// ---- VISUs/PAGE_MAIN.TcVIS
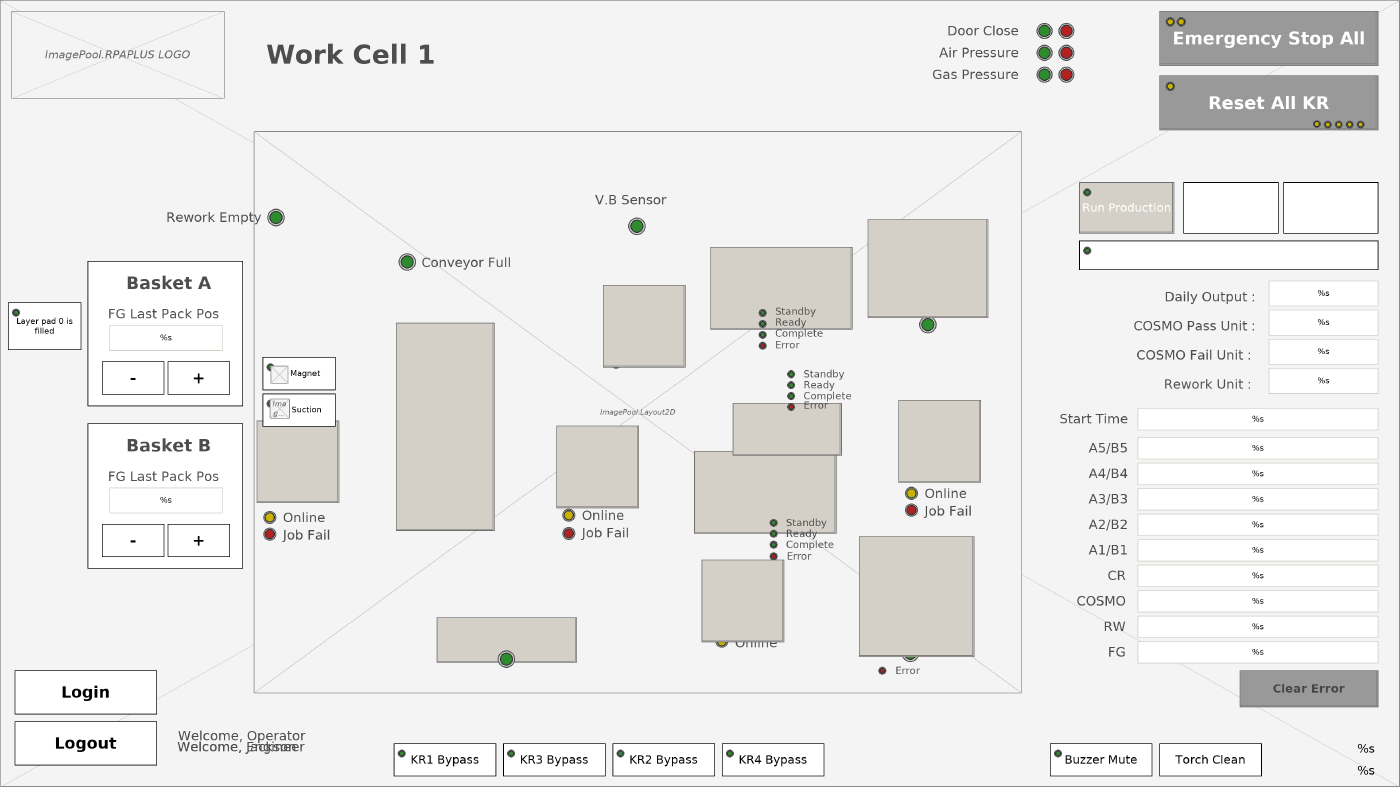
VISUALIZATION PAGE_MAIN  // 1920x1080
    Image (0,0 1920x1080), image: ImagePool.The-New-Silver-Backgrounds
    Frame (0,930 1920x150)
        shows Footer_Main()
        shows Footer_1()
    Frame (0,0 1920x225)
        shows Header()
    Label (362,45 650x60), "Work Cell 1"
    RoundedRectangle (1760,250 130x70), "Reset Production"
        OnMouseClick: OpenDialog Dialog=MSG_BOX_RESET, OpenModal=True, OpenCentered=True
    RoundedRectangle (20,990 195x60), "Logout"
        OnMouseClick: VisuUserMgmt Type=Logout
        OnMouseClick: execute {
            LOGFILE( sLogEvent	 := MSG.EVENT_BTN,
            		 sLogComp	 := MSG.COMP_HMI,
            		 sLogAction	 := MSG.ACTION_LOGOUT,
            	 	 logFlag	 := TRUE);
        }
    RoundedRectangle (20,920 195x60), "Login"
        tap MAIN.BTN_LOG
        OnMouseClick: VisuUserMgmt Type=Login
        OnMouseClick: execute {
            LOGFILE( sLogEvent	 := MSG.EVENT_BTN,
            		 sLogComp	 := MSG.COMP_HMI,
            		 sLogAction	 := MSG.ACTION_LOGIN,
            	 	 logFlag	 := TRUE);
        }
    Label (240,1005 200x40), "Welcome, Engineer"
    Label (240,1005 200x40), "Welcome, Jackson"
    Label (241,990 200x40), "Welcome, Operator"
    RoundedRectangle (120,358 213x199)
    Label (170,366 119x45), "Basket A"
    RoundedRectangle (140,496 85x45), "-"
        tap JIG.BasketA_Minus
        OnMouseClick: execute {
            LOGFILE( sLogEvent	 := MSG.EVENT_BTN,
            		 sLogComp	 := MSG.COMP_FG,
            		 sLogAction	 := MSG.ACTION_BSKTA_MINUS,
            	 	 logFlag	 := TRUE);
        }
    RoundedRectangle (230,496 85x45), "+"
        tap JIG.BasketA_Plus
        OnMouseClick: execute {
            LOGFILE( sLogEvent	 := MSG.EVENT_BTN,
            		 sLogComp	 := MSG.COMP_FG,
            		 sLogAction	 := MSG.ACTION_BSKTA_PLUS,
            	 	 logFlag	 := TRUE);
        }
    Textfield (150,446 155x35), "%s", text variable: GVL.Basket_A_Counter
    Label (145,416 173x30), "FG Last Pack Pos"
    RoundedRectangle (120,581 213x199)
    Label (170,589 119x45), "Basket B"
    RoundedRectangle (140,719 85x45), "-"
        tap JIG.BasketB_Minus
        OnMouseClick: execute {
            LOGFILE( sLogEvent	 := MSG.EVENT_BTN,
            		 sLogComp	 := MSG.COMP_FG,
            		 sLogAction	 := MSG.ACTION_BSKTA_MINUS,
            	 	 logFlag	 := TRUE);
        }
    RoundedRectangle (230,719 85x45), "+"
        tap JIG.BasketB_Plus
        OnMouseClick: execute {
            LOGFILE( sLogEvent	 := MSG.EVENT_BTN,
            		 sLogComp	 := MSG.COMP_FG,
            		 sLogAction	 := MSG.ACTION_BSKTB_PLUS,
            	 	 logFlag	 := TRUE);
        }
    Textfield (150,669 155x35), "%s", text variable: GVL.Basket_B_Counter
    Label (145,639 173x30), "FG Last Pack Pos"
    Image (348,180 1053x771), image: ImagePool.Layout2D
    Lamp1 (865,430 27x27), variable: KR3.bInBit[1,6], style: Lamp-Lamp1-Green
    Lamp1 (1010,815 27x27), variable: KR4.bInBit[1,6], style: Lamp-Lamp1-Green
    Lamp1 (1275,600 27x27), variable: KR5.bInBit[1,6], style: Lamp-Lamp1-Green
    Lamp1 (800,625 27x27), variable: KR2.bInBit[1,6], style: Lamp-Lamp1-Green
    Lamp1 (360,700 20x20), variable: KR1.KROnline, style: Lamp-Lamp1-Yellow
    Button (543,443 135x285)
        OnMouseClick: change screen: PAGE_CoolRack
        OnMouseClick: execute {
            LOGFILE( sLogEvent	 := MSG.EVENT_PAGE,
            		 sLogComp	 := MSG.COMP_CR,
            		 sLogAction	 := MSG.ACTION_COOLRACK,
            	 	 logFlag	 := TRUE);
        }
    Button (599,847 192x62)
        OnMouseClick: change screen: PAGE_COSMO
        OnMouseClick: execute {
            LOGFILE( sLogEvent	 := MSG.EVENT_PAGE,
            		 sLogComp	 := MSG.COMP_CM,
            		 sLogAction	 := MSG.ACTION_COSMO,
            	 	 logFlag	 := TRUE);
        }
    Lamp1 (681,891 27x27), variable: GVL.COSMO_Ready, style: Lamp-Lamp1-Green
    Lamp1 (860,297 27x27), variable: GVL.VibBowl_Ready, style: Lamp-Lamp1-Green
    Label (813,252 255x45), "V.B Sensor"
    Lamp1 (1259,432 27x27), variable: INFEED_RACK.IFRack_Ready, style: Lamp-Lamp1-Green
    Lamp1 (1235,883 27x27), variable: GVL.JIGC_Standby, style: Lamp-Lamp1-Green
    Button (1178,736 158x165)
        OnMouseClick: change screen: PAGE_TTorch
        OnMouseClick: execute {
            LOGFILE( sLogEvent	 := MSG.EVENT_PAGE,
            		 sLogComp	 := MSG.COMP_TT,
            		 sLogAction	 := MSG.ACTION_TT,
            	 	 logFlag	 := TRUE);
        }
    Button (974,339 195x113)
        OnMouseClick: change screen: PAGE_JIG_A
        OnMouseClick: execute {
            LOGFILE( sLogEvent	 := MSG.EVENT_PAGE,
            		 sLogComp	 := MSG.COMP_JIGA,
            		 sLogAction	 := MSG.ACTION_JIGA,
            	 	 logFlag	 := TRUE);
        }
    Button (952,619 195x113)
        OnMouseClick: change screen: PAGE_JIG_C
        OnMouseClick: execute {
            LOGFILE( sLogEvent	 := MSG.EVENT_PAGE,
            		 sLogComp	 := MSG.COMP_JIGC,
            		 sLogAction	 := MSG.ACTION_JIGC,
            	 	 logFlag	 := TRUE);
        }
    Button (1005,553 149x72)
        OnMouseClick: change screen: PAGE_JIG_B
        OnMouseClick: execute {
            LOGFILE( sLogEvent	 := MSG.EVENT_PAGE,
            		 sLogComp	 := MSG.COMP_JIGB,
            		 sLogAction	 := MSG.ACTION_JIGB,
            	 	 logFlag	 := TRUE);
        }
    Lamp1 (365,285 27x27), variable: GVL.Rework_Empty, style: Lamp-Lamp1-Green
    Lamp1 (545,346 27x27), variable: GVL.Conveyor_Full, style: Lamp-Lamp1-Green
    Label (225,276 146x45), "Rework Empty"
    Label (575,338 130x45), "Conveyor Full"
    Lamp1 (360,723 20x20), variable: KR1.bInBit[4,0], style: Lamp-Lamp1-Red
    Lamp1 (1240,690 20x20), variable: KR5.bInBit[4,7], style: Lamp-Lamp1-Red
    Lamp1 (770,722 20x20), variable: KR2.bInBit[3,4], style: Lamp-Lamp1-Red
    Lamp1 (395,633 27x27), variable: KR1.bInBit[1,6], style: Lamp-Lamp1-Green
    Label (385,722 80x25), "Job Fail"
    Label (385,698 80x25), "Online"
    Lamp1 (770,697 20x20), variable: KR2.KROnline, style: Lamp-Lamp1-Yellow
    Label (795,719 80x25), "Job Fail"
    Label (795,695 80x25), "Online"
    Lamp1 (1240,667 20x20), variable: KR5.KROnline, style: Lamp-Lamp1-Yellow
    Label (1265,689 80x25), "Job Fail"
    Label (1265,665 80x25), "Online"
    Lamp1 (835,487 20x20), variable: KR3.KROnline, style: Lamp-Lamp1-Yellow
    Label (860,485 80x25), "Online"
    Lamp1 (980,870 20x20), variable: KR4.KROnline, style: Lamp-Lamp1-Yellow
    Label (1005,870 80x25), "Online"
    Button (827,391 113x113)
        OnMouseClick: change screen: PAGE_KR3
        OnMouseClick: execute {
            LOGFILE( sLogEvent	 := MSG.EVENT_PAGE,
            		 sLogComp	 := MSG.COMP_KR3,
            		 sLogAction	 := MSG.ACTION_KR3,
            	 	 logFlag	 := TRUE);
        }
    Button (763,584 113x113)
        OnMouseClick: change screen: PAGE_KR2
        OnMouseClick: execute {
            LOGFILE( sLogEvent	 := MSG.EVENT_PAGE,
            		 sLogComp	 := MSG.COMP_KR2,
            		 sLogAction	 := MSG.ACTION_KR2,
            	 	 logFlag	 := TRUE);
        }
    Button (962,768 113x113)
        OnMouseClick: change screen: PAGE_KR4
        OnMouseClick: execute {
            LOGFILE( sLogEvent	 := MSG.EVENT_PAGE,
            		 sLogComp	 := MSG.COMP_KR4,
            		 sLogAction	 := MSG.ACTION_KR4,
            	 	 logFlag	 := TRUE);
        }
    Button (1232,549 113x113)
        OnMouseClick: change screen: PAGE_KR5
        OnMouseClick: execute {
            LOGFILE( sLogEvent	 := MSG.EVENT_PAGE,
            		 sLogComp	 := MSG.COMP_KR5,
            		 sLogAction	 := MSG.ACTION_KR5,
            	 	 logFlag	 := TRUE);
        }
    Button (352,577 113x113)
        OnMouseClick: change screen: PAGE_KR1_Tab
        OnMouseClick: execute {
            LOGFILE( sLogEvent	 := MSG.EVENT_PAGE,
            		 sLogComp	 := MSG.COMP_KR1,
            		 sLogAction	 := MSG.ACTION_KR1,
            	 	 logFlag	 := TRUE);
        }
    Label (1500,425 225x45), "COSMO Pass Unit :"
    Textfield (1740,425 150x35), "%s", text variable: GVL.Pass_Counter
    Textfield (1740,465 150x35), "%s", text variable: GVL.Fail_Counter
    Label (1500,465 225x45), "COSMO Fail Unit :"
    Textfield (1560,880 330x30), "%s", text variable: AUTO_MODE.processnameFG
    Group (1430,705 460x30)
        Textfield (130,0 330x30), "%s", text variable: AUTO_MODE.processnameA2
        Label (0,0 120x30), "A2/B2"
    Group (1430,740 460x30)
        Textfield (130,0 330x30), "%s", text variable: AUTO_MODE.processnameA1
        Label (0,0 120x30), "A1/B1"
    Textfield (1560,600 330x30), "%s", text variable: AUTO_MODE.processnameA5
    Label (1430,600 120x30), "A5/B5"
    Group (1430,635 460x30)
        Textfield (130,0 330x30), "%s", text variable: AUTO_MODE.processnameA4
        Label (0,0 120x30), "A4/B4"
    Group (1430,670 460x30)
        Textfield (130,0 330x30), "%s", text variable: AUTO_MODE.processnameA3
        Label (0,0 120x30), "A3/B3"
    Label (1472,880 75x30), "FG"
    Group (1472,845 418x30)
        Textfield (88,0 330x30), "%s", text variable: AUTO_MODE.processnameRW
        Label (0,0 75x30), "RW"
    Group (1472,775 418x30)
        Textfield (88,0 330x30), "%s", text variable: AUTO_MODE.processnameCR
        Label (0,0 75x30), "CR"
    Group (1455,810 435x30)
        Textfield (105,0 330x30), "%s", text variable: AUTO_MODE.processnameCOSMO
        Label (0,0 92x30), "COSMO"
    Lamp1 (1260,358 20x20), variable: INFEED_RACK.IFRack_Ready, style: Lamp-Lamp1-Yellow
    Button (1190,301 165x135)
        OnMouseClick: change screen: PAGE_InfeedRack
        OnMouseClick: execute {
            LOGFILE( sLogEvent	 := MSG.EVENT_PAGE,
            		 sLogComp	 := MSG.COMP_IR,
            		 sLogAction	 := MSG.ACTION_INFEEDRACK,
            	 	 logFlag	 := TRUE);
        }
    Label (1500,385 225x45), "Daily Output :"
    Textfield (1740,385 150x35), "%s", text variable: GVL.daily_output
    Label (1500,505 225x45), "Rework Unit :"
    Textfield (1740,505 150x35), "%s", text variable: GVL.Rework_Counter
    RoundedRectangle (1480,330 410x40), "Welding Mode"
        toggle SAFETY_SENSOR.WELDING_MODE
        OnMouseClick: execute {  }
    RoundedRectangle (1623,250 130x70), "Halt Production", input disabled if: MAIN.btnTorchClean
        OnMouseClick: execute {
            KR1.bOutBit[1,0]:= FALSE;
            KR2.bOutBit[1,0]:= FALSE;
            KR3.bOutBit[1,0]:= FALSE;
            KR4.bOutBit[1,0]:= FALSE;
            KR5.bOutBit[1,0]:= FALSE;
            LOGFILE( sLogEvent	 := MSG.EVENT_BTN,
            		 sLogComp	 := MSG.COMP_HMI,
            		 sLogAction	 := MSG.ACTION_STOP,
            	 	 logFlag	 := TRUE);
            AUTO_MODE.Halt_Production := TRUE;
            AUTO_MODE.AutoMode := False;
        }
    Button (1480,250 130x70), "Run Production", pressed state: AUTO_MODE.AutoMode, input disabled if: MAIN.btnTorchClean
        toggle AUTO_MODE.AutoMode
        OnMouseClick: execute {
            LOGFILE( sLogEvent	 := MSG.EVENT_BTN,
            		 sLogComp	 := MSG.COMP_HMI,
            		 sLogAction	 := MSG.ACTION_START,
            	 	 logFlag	 := TRUE);
            IF AUTO_MODE.AutoMode THEN
            	AUTO_MODE.Start_time := MAIN.fb_TimeStamp.SystemTime;
            END_IF
        }
    Lamp1 (1485,255 12x18), variable: AUTO_MODE.AutoMode, style: Lamp-Lamp1-Green
    Textfield (1560,560 330x30), "%s", text variable: AUTO_MODE.Start_time
    Label (1430,560 120x30), "Start Time"
    Lamp1 (1485,335 12x18), variable: SAFETY_SENSOR.WELDING_MODE, style: Lamp-Lamp1-Green
    Group (1250,20 225x105)
        Group (0,0 225x45)
            Label (0,0 150x45), "Door Close"
            Lamp1 (170,10 25x25), variable: SAFETY_SENSOR.SENSOR_SAFETY_DOOR_CLOSE, style: Lamp-Lamp1-Green
            Lamp1 (200,10 25x25), variable: not SAFETY_SENSOR.SENSOR_SAFETY_DOOR_CLOSE, style: Lamp-Lamp1-Red
        Label (0,30 150x45), "Air Pressure"
        Lamp1 (170,40 25x25), variable: SAFETY_SENSOR.SENSOR_AIR_PRESSURE_OK, style: Lamp-Lamp1-Green
        Lamp1 (200,40 25x25), variable: not SAFETY_SENSOR.SENSOR_AIR_PRESSURE_OK or SAFETY_SENSOR.SENSOR_AIR_PRESSURE_HIGH, style: Lamp-Lamp1-Red
        Label (0,60 150x45), "Gas Pressure"
        Lamp1 (170,70 25x25), variable: SAFETY_SENSOR.SENSOR_GAS_PRESSURE_OK, style: Lamp-Lamp1-Green
        Lamp1 (200,70 25x25), variable: not SAFETY_SENSOR.SENSOR_GAS_PRESSURE_OK or SAFETY_SENSOR.SENSOR_GAS_PRESSURE_HIGH, style: Lamp-Lamp1-Red
    Group (1079,506 100x45)
        Lamp1 (0,0 12x15), variable: GVL.JIGB_Standby, style: Lamp-Lamp1-Green
        Lamp1 (0,15 12x15), variable: GVL.JIGB_Ready, style: Lamp-Lamp1-Green
        Label (20,0 80x15), "Standby"
        Label (20,15 80x15), "Ready"
        Label (20,30 80x15), "Complete"
        Lamp1 (0,30 12x15), variable: GVL.JIGB_Complete, style: Lamp-Lamp1-Green
    Lamp1 (1040,422 12x15), variable: GVL.JIGA_Standby, style: Lamp-Lamp1-Green
    Lamp1 (1040,437 12x15), variable: GVL.JIGA_Ready, style: Lamp-Lamp1-Green
    Label (1060,420 80x15), "Standby"
    Label (1060,435 80x15), "Ready"
    Label (1060,450 80x15), "Complete"
    Lamp1 (1040,452 12x15), variable: GVL.JIGA_Complete, style: Lamp-Lamp1-Green
    Lamp1 (1055,710 12x15), variable: GVL.JIGC_Standby, style: Lamp-Lamp1-Green
    Lamp1 (1055,725 12x15), variable: GVL.JIGC_Ready, style: Lamp-Lamp1-Green
    Label (1075,710 80x15), "Standby"
    Label (1075,725 80x15), "Ready"
    Label (1075,740 80x15), "Complete"
    Lamp1 (1055,740 12x15), variable: GVL.JIGC_Complete, style: Lamp-Lamp1-Green
    Button (1700,920 190x50), "Clear Error", pressed state: MAIN.btn_Reset or MAIN.Reset_State
        toggle GVL.ClearError
        OnMouseClick: execute {
            LOGFILE( sLogEvent	 := MSG.EVENT_BTN,
            		 sLogComp	 := MSG.COMP_HMI,
            		 sLogAction	 := MSG.ACTION_CLEAR_ERROR,
            	 	 logFlag	 := TRUE);
        }
    Label (1060,466 80x15), "Error"
    Lamp1 (1040,467 12x15), variable: AUTO_MODE.JIGA_ErrorState, style: Lamp-Lamp1-Red
    Lamp1 (1079,551 12x15), variable: AUTO_MODE.JIGB_ErrorState, style: Lamp-Lamp1-Red
    Label (1099,549 80x15), "Error"
    Lamp1 (1055,756 12x15), variable: AUTO_MODE.JIGC_ErrorState, style: Lamp-Lamp1-Red
    Label (1076,756 80x15), "Error"
    Lamp1 (1204,913 12x15), variable: AUTO_MODE.TT_ErrorState, style: Lamp-Lamp1-Red
    Label (1225,913 80x15), "Error"
    RoundedRectangle (1590,1020 140x45), "Torch Clean"
        toggle MAIN.btnTorchClean
        OnMouseClick: execute {  }
    Group (1440,1020 140x45)
        RoundedRectangle (0,0 140x45), "Buzzer Mute"
            toggle TL.Buzzer_mute
            OnMouseClick: execute {  }
        Lamp1 (5,5 12x18), variable: TL.Buzzer_mute, style: Lamp-Lamp1-Green
    Group (840,1020 290x45)
        Group (150,0 140x45)
            RoundedRectangle (0,0 140x45), "KR4 Bypass"
                OnMouseClick: OpenDialog Dialog=MSG_KR4_BP, OpenModal=True, OpenCentered=True
            Lamp1 (5,5 12x18), variable: GVL.KR4_bypass, style: Lamp-Lamp1-Green
        RoundedRectangle (0,0 140x45), "KR2 Bypass"
            OnMouseClick: OpenDialog Dialog=MSG_KR2_BP, OpenModal=True, OpenCentered=True
        Lamp1 (5,5 12x18), variable: GVL.KR2_bypass, style: Lamp-Lamp1-Green
    RoundedRectangle (690,1020 140x45), "KR3 Bypass"
        OnMouseClick: OpenDialog Dialog=MSG_KR3_BP, OpenModal=True, OpenCentered=True
    Lamp1 (695,1025 12x18), variable: GVL.KR3_bypass, style: Lamp-Lamp1-Green
    RoundedRectangle (540,1020 140x45), "KR1 Bypass"
        OnMouseClick: OpenDialog Dialog=MSG_KR1_BP, OpenModal=True, OpenCentered=True
    Lamp1 (545,1025 12x18), variable: GVL.KR1_bypass, style: Lamp-Lamp1-Green
    Group (360,490 100x45)
        RoundedRectangle (0,0 100x45), "Magnet"
            OnMouseClick: OpenDialog Dialog=MSG_EOAT, OpenModal=True, OpenCentered=True
        Lamp1 (5,5 12x18), variable: GVL.KR1_EOAT_FILL, style: Lamp-Lamp1-Green
        Image (11,12 24x24), image: ImagePool.001-resources
    Group (360,540 100x45)
        RoundedRectangle (0,0 100x45), "Suction"
            OnMouseClick: OpenDialog Dialog=MSG_EOAT_SUCTION, OpenModal=True, OpenCentered=True
        Lamp1 (5,5 12x18), variable: GVL.KR1_EOAT_SUCTION, style: Lamp-Lamp1-Green
        Image (10,7 27x27), angle 180, image: ImagePool.002-plunger
    RoundedRectangle (11,415 100x65), "Layer pad 0 is filled"
        toggle GVL.LAYERPAD0
    Lamp1 (16,420 12x18), variable: GVL.LAYERPAD0, style: Lamp-Lamp1-Green
END_VISUALIZATION

// ---- VISUs/PAGE_KR2.TcVIS
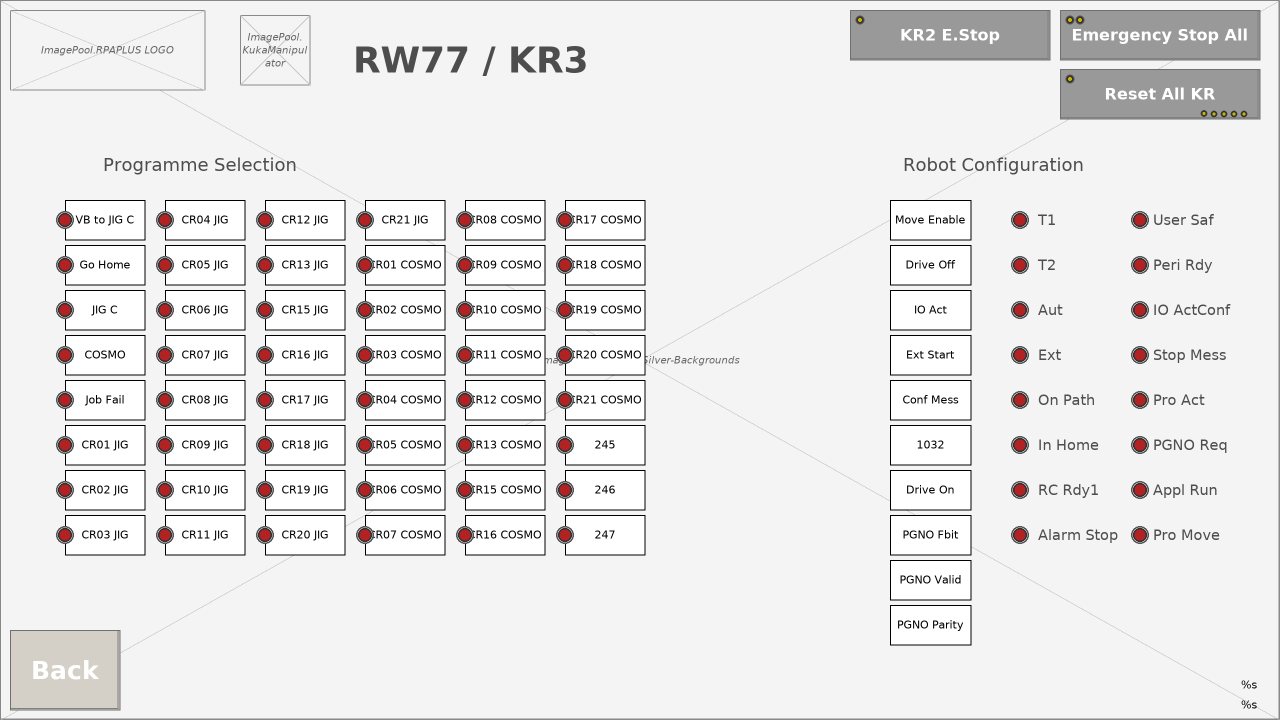
VISUALIZATION PAGE_KR2  // 1280x720
    Image (0,0 1280x720), image: ImagePool.The-New-Silver-Backgrounds
    Frame (0,620 1280x100)
        shows Footer_Back()
    Frame (0,0 1280x150)
        shows Header()
    Label (350,40 300x40), "RW77 / KR3"
    Label (100,150 250x30), "Programme Selection"
    Group (850,10 200x50)
        Button (0,0 200x50), "KR2 E.Stop"
            toggle KR2.KR2_Estop
        Lamp1 (5,5 10x10), variable: KR2.KR2_Estop, style: Lamp-Lamp1-Yellow
    Image (240,15 70x70), image: ImagePool.KukaManipulator
    Label (900,150 200x30), "Robot Configuration"
    RoundedRectangle (890,200 81x40), "Move Enable"
        toggle KR2.bOutBit[1,0]
    RoundedRectangle (890,245 81x40), "Drive Off"
        toggle KR2.bOutBit[1,1]
    RoundedRectangle (890,290 81x40), "IO Act"
        toggle KR2.bOutBit[1,2]
    RoundedRectangle (890,335 81x40), "Ext Start"
        toggle KR2.bOutBit[1,3]
    RoundedRectangle (890,380 81x40), "Conf Mess"
        toggle KR2.bOutBit[1,4]
    RoundedRectangle (890,425 81x40), "1032"
        toggle KR2.bOutBit[1,5]
    RoundedRectangle (890,470 81x40), "Drive On"
        toggle KR2.bOutBit[1,6]
    RoundedRectangle (890,515 81x40), "PGNO Fbit"
        toggle KR2.bOutBit[1,7]
    RoundedRectangle (890,560 81x40), "PGNO Valid"
        toggle KR2.bOutBit[2,0]
    RoundedRectangle (890,605 81x40), "PGNO Parity"
        toggle KR2.bOutBit[2,1]
    Label (1150,205 110x30), "User Saf"
    Label (1150,250 110x30), "Peri Rdy"
    Label (1150,295 110x30), "IO ActConf"
    Label (1150,340 110x30), "Stop Mess"
    Label (1150,385 110x30), "Pro Act"
    Label (1150,430 110x30), "PGNO Req"
    Label (1150,475 110x30), "Appl Run"
    Label (1150,520 110x30), "Pro Move"
    Label (1035,205 105x30), "T1"
    Label (1035,250 105x30), "T2"
    Label (1035,295 105x30), "Aut"
    Label (1035,340 105x30), "Ext"
    Label (1035,385 105x30), "On Path"
    Label (1035,430 105x30), "In Home"
    Label (1035,475 105x30), "RC Rdy1"
    Label (1035,520 105x30), "Alarm Stop"
    Lamp1 (1010,210 20x20), variable: KR2.bInBit[1,0], style: Lamp-Lamp1-Red
    Lamp1 (1010,255 20x20), variable: KR2.bInBit[1,1], style: Lamp-Lamp1-Red
    Lamp1 (1010,300 20x20), variable: KR2.bInBit[1,2], style: Lamp-Lamp1-Red
    Lamp1 (1010,345 20x20), variable: KR2.bInBit[1,3], style: Lamp-Lamp1-Red
    Lamp1 (1010,390 20x20), variable: KR2.bInBit[1,4], style: Lamp-Lamp1-Red
    Lamp1 (1010,435 20x20), variable: KR2.bInBit[1,5], style: Lamp-Lamp1-Red
    Lamp1 (1010,480 20x20), variable: KR2.bInBit[1,6], style: Lamp-Lamp1-Red
    Lamp1 (1010,525 20x20), variable: KR2.bInBit[1,7], style: Lamp-Lamp1-Red
    Lamp1 (1130,210 20x20), variable: KR2.bInBit[2,0], style: Lamp-Lamp1-Red
    Lamp1 (1130,255 20x20), variable: KR2.bInBit[2,1], style: Lamp-Lamp1-Red
    Lamp1 (1130,300 20x20), variable: KR2.bInBit[2,2], style: Lamp-Lamp1-Red
    Lamp1 (1130,345 20x20), variable: KR2.bInBit[2,3], style: Lamp-Lamp1-Red
    Lamp1 (1130,390 20x20), variable: KR2.bInBit[2,4], style: Lamp-Lamp1-Red
    Lamp1 (1130,435 20x20), variable: KR2.bInBit[2,5], style: Lamp-Lamp1-Red
    Lamp1 (1130,480 20x20), variable: KR2.bInBit[2,6], style: Lamp-Lamp1-Red
    Lamp1 (1130,525 20x20), variable: KR2.bInBit[2,7], style: Lamp-Lamp1-Red
    RoundedRectangle (65,200 80x40), "VB to JIG C"
        toggle KR2.bOutBit[3,0]
    RoundedRectangle (65,245 80x40), "Go Home"
        toggle KR2.bOutBit[3,1]
    RoundedRectangle (65,290 80x40), "JIG C"
        toggle KR2.bOutBit[3,2]
    RoundedRectangle (65,335 80x40), "COSMO"
        toggle KR2.bOutBit[3,3]
    RoundedRectangle (65,380 80x40), "Job Fail"
        toggle KR2.bOutBit[3,4]
    RoundedRectangle (65,425 80x40), "CR01 JIG"
        toggle KR2.bOutBit[3,5]
    RoundedRectangle (65,470 80x40), "CR02 JIG"
        toggle KR2.bOutBit[3,6]
    RoundedRectangle (65,515 80x40), "CR03 JIG"
        toggle KR2.bOutBit[3,7]
    Lamp1 (55,210 20x20), variable: KR2.bInBit[3,0], style: Lamp-Lamp1-Red
    Lamp1 (55,255 20x20), variable: KR2.bInBit[3,1], style: Lamp-Lamp1-Red
    Lamp1 (55,300 20x20), variable: KR2.bInBit[3,2], style: Lamp-Lamp1-Red
    Lamp1 (55,345 20x20), variable: KR2.bInBit[3,3], style: Lamp-Lamp1-Red
    Lamp1 (55,390 20x20), variable: KR2.bInBit[3,4], style: Lamp-Lamp1-Red
    Lamp1 (55,435 20x20), variable: KR2.bInBit[3,5], style: Lamp-Lamp1-Red
    Lamp1 (55,480 20x20), variable: KR2.bInBit[3,6], style: Lamp-Lamp1-Red
    Lamp1 (55,525 20x20), variable: KR2.bInBit[3,7], style: Lamp-Lamp1-Red
    RoundedRectangle (265,200 80x40), "CR12 JIG"
        toggle KR2.bOutBit[5,0]
    RoundedRectangle (265,245 80x40), "CR13 JIG"
        toggle KR2.bOutBit[5,1]
    RoundedRectangle (265,290 80x40), "CR15 JIG"
        toggle KR2.bOutBit[5,2]
    RoundedRectangle (265,335 80x40), "CR16 JIG"
        toggle KR2.bOutBit[5,3]
    RoundedRectangle (265,380 80x40), "CR17 JIG"
        toggle KR2.bOutBit[5,4]
    RoundedRectangle (265,425 80x40), "CR18 JIG"
        toggle KR2.bOutBit[5,5]
    RoundedRectangle (265,470 80x40), "CR19 JIG"
        toggle KR2.bOutBit[5,6]
    RoundedRectangle (265,515 80x40), "CR20 JIG"
        toggle KR2.bOutBit[5,7]
    Lamp1 (255,210 20x20), variable: KR2.bInBit[5,0], style: Lamp-Lamp1-Red
    Lamp1 (255,255 20x20), variable: KR2.bInBit[5,1], style: Lamp-Lamp1-Red
    Lamp1 (255,300 20x20), variable: KR2.bInBit[5,2], style: Lamp-Lamp1-Red
    Lamp1 (255,345 20x20), variable: KR2.bInBit[5,3], style: Lamp-Lamp1-Red
    Lamp1 (255,390 20x20), variable: KR2.bInBit[5,4], style: Lamp-Lamp1-Red
    Lamp1 (255,435 20x20), variable: KR2.bInBit[5,5], style: Lamp-Lamp1-Red
    Lamp1 (255,480 20x20), variable: KR2.bInBit[5,6], style: Lamp-Lamp1-Red
    Lamp1 (255,525 20x20), variable: KR2.bInBit[5,7], style: Lamp-Lamp1-Red
    RoundedRectangle (365,200 80x40), "CR21 JIG"
        toggle KR2.bOutBit[6,0]
    RoundedRectangle (365,245 80x40), "CR01 COSMO"
        toggle KR2.bOutBit[6,1]
    RoundedRectangle (365,290 80x40), "CR02 COSMO"
        toggle KR2.bOutBit[6,2]
    RoundedRectangle (365,335 80x40), "CR03 COSMO"
        toggle KR2.bOutBit[6,3]
    RoundedRectangle (365,380 80x40), "CR04 COSMO"
        toggle KR2.bOutBit[6,4]
    RoundedRectangle (365,425 80x40), "CR05 COSMO"
        toggle KR2.bOutBit[6,5]
    RoundedRectangle (365,470 80x40), "CR06 COSMO"
        toggle KR2.bOutBit[6,6]
    RoundedRectangle (365,515 80x40), "CR07 COSMO"
        toggle KR2.bOutBit[6,7] p2164770859=TRUE
    Lamp1 (355,210 20x20), variable: KR2.bInBit[6,0], style: Lamp-Lamp1-Red
    Lamp1 (355,255 20x20), variable: KR2.bInBit[6,1], style: Lamp-Lamp1-Red
    Lamp1 (355,300 20x20), variable: KR2.bInBit[6,2], style: Lamp-Lamp1-Red
    Lamp1 (355,345 20x20), variable: KR2.bInBit[6,3], style: Lamp-Lamp1-Red
    Lamp1 (355,390 20x20), variable: KR2.bInBit[6,4], style: Lamp-Lamp1-Red
    Lamp1 (355,435 20x20), variable: KR2.bInBit[6,5], style: Lamp-Lamp1-Red
    Lamp1 (355,480 20x20), variable: KR2.bInBit[6,6], style: Lamp-Lamp1-Red
    Lamp1 (355,525 20x20), variable: KR2.bInBit[6,7], style: Lamp-Lamp1-Red
    RoundedRectangle (465,200 80x40), "CR08 COSMO"
        toggle KR2.bOutBit[7,0]
    RoundedRectangle (465,245 80x40), "CR09 COSMO"
        toggle KR2.bOutBit[7,1]
    RoundedRectangle (465,290 80x40), "CR10 COSMO"
        toggle KR2.bOutBit[7,2]
    RoundedRectangle (465,335 80x40), "CR11 COSMO"
        toggle KR2.bOutBit[7,3]
    RoundedRectangle (465,380 80x40), "CR12 COSMO"
        toggle KR2.bOutBit[7,4]
    RoundedRectangle (465,425 80x40), "CR13 COSMO"
        toggle KR2.bOutBit[7,5]
    RoundedRectangle (465,470 80x40), "CR15 COSMO"
        toggle KR2.bOutBit[7,6]
    RoundedRectangle (465,515 80x40), "CR16 COSMO"
        toggle KR2.bOutBit[7,7] p2164770859=TRUE
    Lamp1 (455,210 20x20), variable: KR2.bInBit[7,0], style: Lamp-Lamp1-Red
    Lamp1 (455,255 20x20), variable: KR2.bInBit[7,1], style: Lamp-Lamp1-Red
    Lamp1 (455,300 20x20), variable: KR2.bInBit[7,2], style: Lamp-Lamp1-Red
    Lamp1 (455,345 20x20), variable: KR2.bInBit[7,3], style: Lamp-Lamp1-Red
    Lamp1 (455,390 20x20), variable: KR2.bInBit[7,4], style: Lamp-Lamp1-Red
    Lamp1 (455,435 20x20), variable: KR2.bInBit[7,5], style: Lamp-Lamp1-Red
    Lamp1 (455,480 20x20), variable: KR2.bInBit[7,6], style: Lamp-Lamp1-Red
    Lamp1 (455,525 20x20), variable: KR2.bInBit[7,7], style: Lamp-Lamp1-Red
    RoundedRectangle (565,200 80x40), "CR17 COSMO"
        toggle KR2.bOutBit[8,0]
    RoundedRectangle (565,245 80x40), "CR18 COSMO"
        toggle KR2.bOutBit[8,1]
    RoundedRectangle (565,290 80x40), "CR19 COSMO"
        toggle KR2.bOutBit[8,2]
    RoundedRectangle (565,335 80x40), "CR20 COSMO"
        toggle KR2.bOutBit[8,3]
    RoundedRectangle (565,380 80x40), "CR21 COSMO"
        toggle KR2.bOutBit[8,4]
    RoundedRectangle (565,425 80x40), "245"
        toggle KR2.bOutBit[8,5]
    RoundedRectangle (565,470 80x40), "246"
        toggle KR2.bOutBit[8,6]
    RoundedRectangle (565,515 80x40), "247"
        toggle KR2.bOutBit[8,7] p2164770859=TRUE
    Lamp1 (555,210 20x20), variable: KR2.bInBit[8,0], style: Lamp-Lamp1-Red
    Lamp1 (555,255 20x20), variable: KR2.bInBit[8,1], style: Lamp-Lamp1-Red
    Lamp1 (555,300 20x20), variable: KR2.bInBit[8,2], style: Lamp-Lamp1-Red
    Lamp1 (555,345 20x20), variable: KR2.bInBit[8,3], style: Lamp-Lamp1-Red
    Lamp1 (555,390 20x20), variable: KR2.bInBit[8,4], style: Lamp-Lamp1-Red
    Lamp1 (555,435 20x20), variable: KR2.bInBit[8,5], style: Lamp-Lamp1-Red
    Lamp1 (555,480 20x20), variable: KR2.bInBit[8,6], style: Lamp-Lamp1-Red
    Lamp1 (555,525 20x20), variable: KR2.bInBit[8,7], style: Lamp-Lamp1-Red
    RoundedRectangle (165,200 80x40), "CR04 JIG"
        toggle KR2.bOutBit[4,0]
    RoundedRectangle (165,245 80x40), "CR05 JIG"
        toggle KR2.bOutBit[4,1]
    RoundedRectangle (165,290 80x40), "CR06 JIG"
        toggle KR2.bOutBit[4,2]
    RoundedRectangle (165,335 80x40), "CR07 JIG"
        toggle KR2.bOutBit[4,3]
    RoundedRectangle (165,380 80x40), "CR08 JIG"
        toggle KR2.bOutBit[4,4]
    RoundedRectangle (165,425 80x40), "CR09 JIG"
        toggle KR2.bOutBit[4,5]
    RoundedRectangle (165,470 80x40), "CR10 JIG"
        toggle KR2.bOutBit[4,6]
    RoundedRectangle (165,515 80x40), "CR11 JIG"
        toggle KR2.bOutBit[4,7]
    Lamp1 (155,210 20x20), variable: KR2.bInBit[4,0], style: Lamp-Lamp1-Red
    Lamp1 (155,255 20x20), variable: KR2.bInBit[4,1], style: Lamp-Lamp1-Red
    Lamp1 (155,300 20x20), variable: KR2.bInBit[4,2], style: Lamp-Lamp1-Red
    Lamp1 (155,345 20x20), variable: KR2.bInBit[4,3], style: Lamp-Lamp1-Red
    Lamp1 (155,390 20x20), variable: KR2.bInBit[4,4], style: Lamp-Lamp1-Red
    Lamp1 (155,435 20x20), variable: KR2.bInBit[4,5], style: Lamp-Lamp1-Red
    Lamp1 (155,480 20x20), variable: KR2.bInBit[4,6], style: Lamp-Lamp1-Red
    Lamp1 (155,525 20x20), variable: KR2.bInBit[4,7], style: Lamp-Lamp1-Red
END_VISUALIZATION

// ---- VISUs/PAGE_KR3.TcVIS
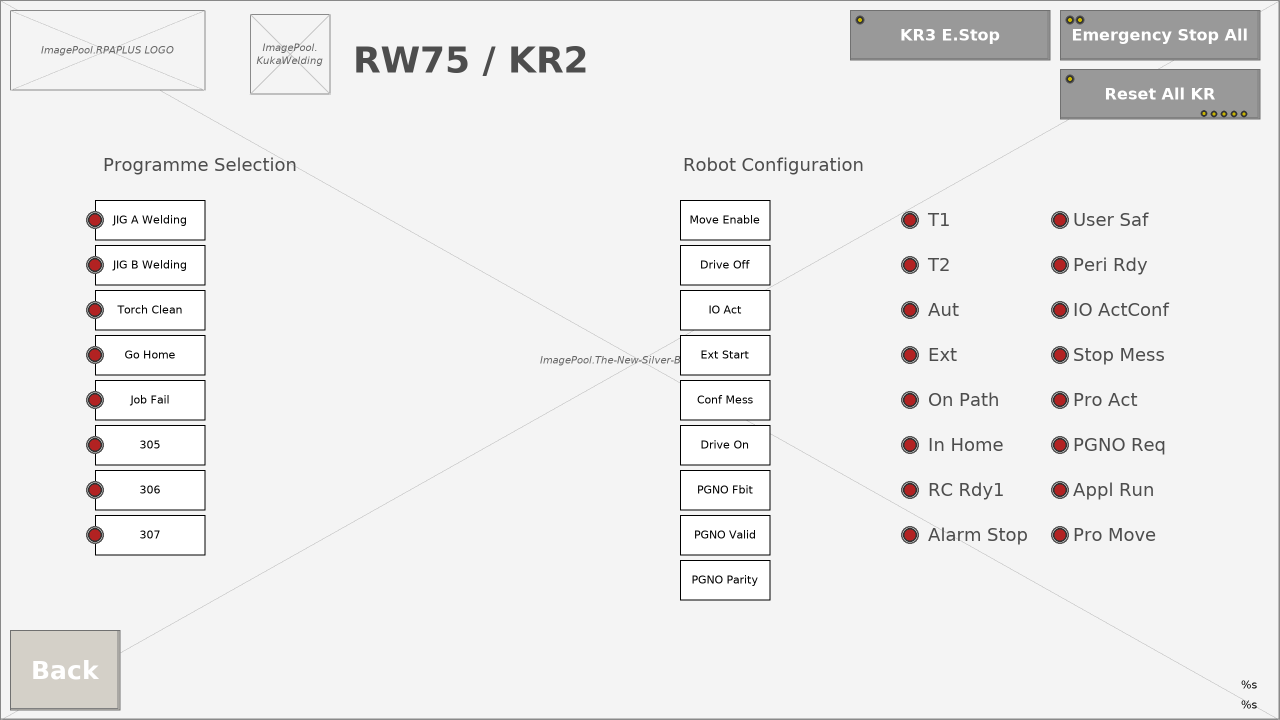
VISUALIZATION PAGE_KR3  // 1280x720
    Image (0,0 1280x720), image: ImagePool.The-New-Silver-Backgrounds
    Frame (0,620 1280x100)
        shows Footer_Back()
    Frame (0,0 1280x150)
        shows Header()
    Image (250,14 80x80), image: ImagePool.KukaWelding
    Label (350,40 300x40), "RW75 / KR2"
    Label (100,150 200x30), "Programme Selection"
    RoundedRectangle (95,200 110x40), "JIG A Welding"
        toggle KR3.bOutBit[3,0]
    RoundedRectangle (95,245 110x40), "JIG B Welding"
        toggle KR3.bOutBit[3,1]
    RoundedRectangle (95,290 110x40), "Torch Clean"
        toggle KR3.bOutBit[3,2]
    RoundedRectangle (95,335 110x40), "Go Home"
        toggle KR3.bOutBit[3,3]
    RoundedRectangle (95,380 110x40), "Job Fail"
        toggle KR3.bOutBit[3,4]
    RoundedRectangle (95,425 110x40), "305"
        toggle KR3.bOutBit[3,5]
    RoundedRectangle (95,470 110x40), "306"
        toggle KR3.bOutBit[3,6]
    RoundedRectangle (95,515 110x40), "307"
        toggle KR3.bOutBit[3,7]
    RoundedRectangle (680,560 90x40), "PGNO Parity"
        toggle KR3.bOutBit[2,0]
    Label (680,150 200x30), "Robot Configuration"
    Lamp1 (85,210 20x20), variable: KR3.bInBit[3,0], style: Lamp-Lamp1-Red
    Lamp1 (85,255 20x20), variable: KR3.bInBit[3,1], style: Lamp-Lamp1-Red
    Lamp1 (85,300 20x20), variable: KR3.bInBit[3,2], style: Lamp-Lamp1-Red
    Lamp1 (85,345 20x20), variable: KR3.bInBit[3,3], style: Lamp-Lamp1-Red
    Lamp1 (85,390 20x20), variable: KR3.bInBit[3,4], style: Lamp-Lamp1-Red
    Lamp1 (85,435 20x20), variable: KR3.bInBit[3,5], style: Lamp-Lamp1-Red
    Lamp1 (85,480 20x20), variable: KR3.bInBit[3,6], style: Lamp-Lamp1-Red
    Lamp1 (85,525 20x20), variable: KR3.bInBit[3,7], style: Lamp-Lamp1-Red
    Lamp1 (900,210 20x20), variable: KR3.bInBit[1,0], style: Lamp-Lamp1-Red
    Lamp1 (900,255 20x20), variable: KR3.bInBit[1,1], style: Lamp-Lamp1-Red
    Lamp1 (900,300 20x20), variable: KR3.bInBit[1,2], style: Lamp-Lamp1-Red
    Lamp1 (900,345 20x20), variable: KR3.bInBit[1,3], style: Lamp-Lamp1-Red
    Lamp1 (900,390 20x20), variable: KR3.bInBit[1,4], style: Lamp-Lamp1-Red
    Lamp1 (900,435 20x20), variable: KR3.bInBit[1,5], style: Lamp-Lamp1-Red
    Lamp1 (900,480 20x20), variable: KR3.bInBit[1,6], style: Lamp-Lamp1-Red
    Lamp1 (900,525 20x20), variable: KR3.bInBit[1,7], style: Lamp-Lamp1-Red
    Lamp1 (1050,210 20x20), variable: KR3.bInBit[2,0], style: Lamp-Lamp1-Red
    Lamp1 (1050,255 20x20), variable: KR3.bInBit[2,1], style: Lamp-Lamp1-Red
    Lamp1 (1050,300 20x20), variable: KR3.bInBit[2,2], style: Lamp-Lamp1-Red
    Lamp1 (1050,345 20x20), variable: KR3.bInBit[2,3], style: Lamp-Lamp1-Red
    Lamp1 (1050,390 20x20), variable: KR3.bInBit[2,4], style: Lamp-Lamp1-Red
    Lamp1 (1050,435 20x20), variable: KR3.bInBit[2,5], style: Lamp-Lamp1-Red
    Lamp1 (1050,480 20x20), variable: KR3.bInBit[2,6], style: Lamp-Lamp1-Red
    Lamp1 (1050,525 20x20), variable: KR3.bInBit[2,7], style: Lamp-Lamp1-Red
    Group (850,10 200x50)
        Button (0,0 200x50), "KR3 E.Stop"
            toggle KR3.KR3_Estop
        Lamp1 (5,5 10x10), variable: KR3.KR3_Estop, style: Lamp-Lamp1-Yellow
    Label (1070,205 110x30), "User Saf"
    Label (1070,250 110x30), "Peri Rdy"
    Label (1070,295 110x30), "IO ActConf"
    Label (1070,340 110x30), "Stop Mess"
    Label (1070,385 110x30), "Pro Act"
    Label (1070,430 110x30), "PGNO Req"
    Label (1070,475 110x30), "Appl Run"
    Label (1070,520 110x30), "Pro Move"
    Label (925,205 105x30), "T1"
    Label (925,250 105x30), "T2"
    Label (925,295 105x30), "Aut"
    Label (925,340 105x30), "Ext"
    Label (925,385 105x30), "On Path"
    Label (925,430 105x30), "In Home"
    Label (925,475 105x30), "RC Rdy1"
    Label (925,520 105x30), "Alarm Stop"
    RoundedRectangle (680,200 90x40), "Move Enable"
        toggle KR3.bOutBit[1,0]
    RoundedRectangle (680,245 90x40), "Drive Off"
        toggle KR3.bOutBit[1,1]
    RoundedRectangle (680,290 90x40), "IO Act"
        toggle KR3.bOutBit[1,2]
    RoundedRectangle (680,335 90x40), "Ext Start"
        toggle KR3.bOutBit[1,3]
    RoundedRectangle (680,380 90x40), "Conf Mess"
        toggle KR3.bOutBit[1,4]
    RoundedRectangle (680,425 90x40), "Drive On"
        toggle KR3.bOutBit[1,5]
    RoundedRectangle (680,470 90x40), "PGNO Fbit"
        toggle KR3.bOutBit[1,6]
    RoundedRectangle (680,515 90x40), "PGNO Valid"
        toggle KR3.bOutBit[1,7]
END_VISUALIZATION

// ---- VISUs/PAGE_KR4.TcVIS
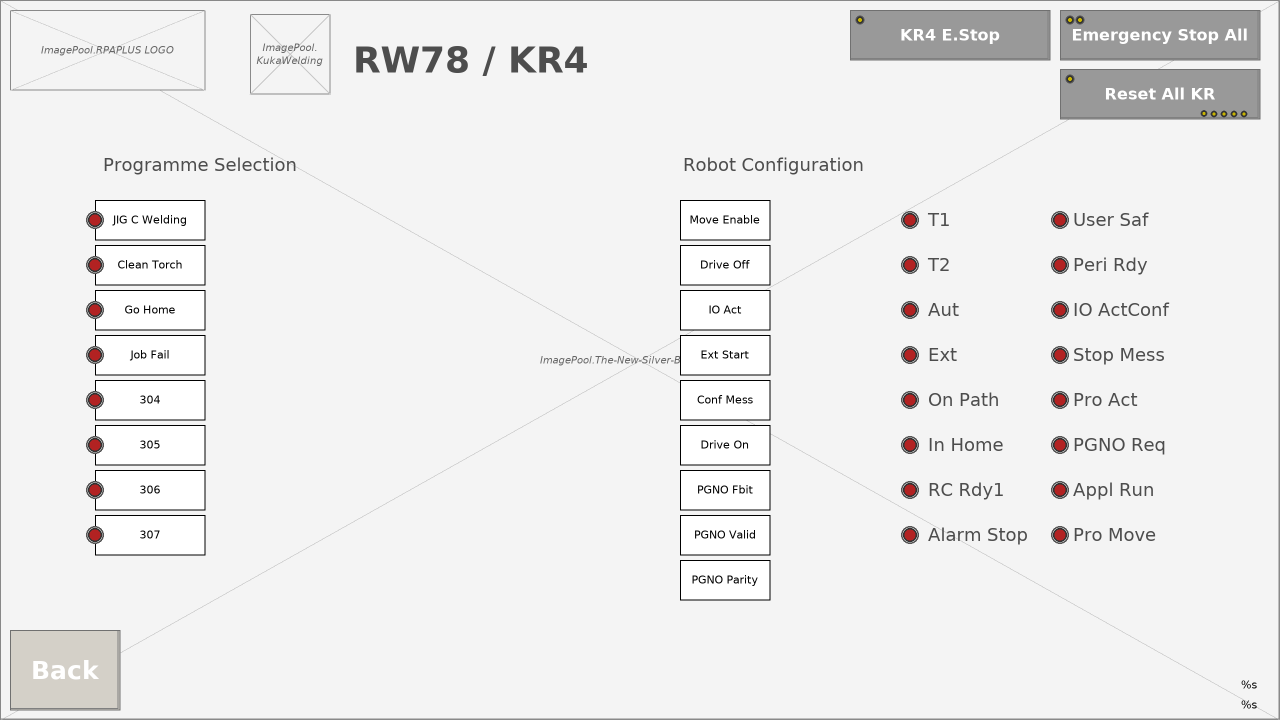
VISUALIZATION PAGE_KR4  // 1280x720
    Image (0,0 1280x720), image: ImagePool.The-New-Silver-Backgrounds
    Frame (0,620 1280x100)
        shows Footer_Back()
    Frame (0,0 1280x150)
        shows Header()
    Image (250,14 80x80), image: ImagePool.KukaWelding
    Label (350,40 300x40), "RW78 / KR4"
    Label (100,150 200x30), "Programme Selection"
    RoundedRectangle (680,200 90x40), "Move Enable"
        toggle KR4.bOutBit[1,0]
    RoundedRectangle (680,245 90x40), "Drive Off"
        toggle KR4.bOutBit[1,1]
    RoundedRectangle (680,290 90x40), "IO Act"
        toggle KR4.bOutBit[1,2]
    RoundedRectangle (680,335 90x40), "Ext Start"
        toggle KR4.bOutBit[1,3]
    RoundedRectangle (680,380 90x40), "Conf Mess"
        toggle KR4.bOutBit[1,4]
    RoundedRectangle (680,425 90x40), "Drive On"
        toggle KR4.bOutBit[1,5]
    RoundedRectangle (680,470 90x40), "PGNO Fbit"
        toggle KR4.bOutBit[1,6]
    RoundedRectangle (680,515 90x40), "PGNO Valid"
        toggle KR4.bOutBit[1,7]
    RoundedRectangle (680,560 90x40), "PGNO Parity"
        toggle KR4.bOutBit[2,0]
    Label (680,150 200x30), "Robot Configuration"
    Lamp1 (900,210 20x20), variable: KR4.bInBit[1,0], style: Lamp-Lamp1-Red
    Lamp1 (900,255 20x20), variable: KR4.bInBit[1,1], style: Lamp-Lamp1-Red
    Lamp1 (900,300 20x20), variable: KR4.bInBit[1,2], style: Lamp-Lamp1-Red
    Lamp1 (900,345 20x20), variable: KR4.bInBit[1,3], style: Lamp-Lamp1-Red
    Lamp1 (900,390 20x20), variable: KR4.bInBit[1,4], style: Lamp-Lamp1-Red
    Lamp1 (900,435 20x20), variable: KR4.bInBit[1,5], style: Lamp-Lamp1-Red
    Lamp1 (900,480 20x20), variable: KR4.bInBit[1,6], style: Lamp-Lamp1-Red
    Lamp1 (900,525 20x20), variable: KR4.bInBit[1,7], style: Lamp-Lamp1-Red
    Lamp1 (1050,210 20x20), variable: KR4.bInBit[2,0], style: Lamp-Lamp1-Red
    Lamp1 (1050,255 20x20), variable: KR4.bInBit[2,1], style: Lamp-Lamp1-Red
    Lamp1 (1050,300 20x20), variable: KR4.bInBit[2,2], style: Lamp-Lamp1-Red
    Lamp1 (1050,345 20x20), variable: KR4.bInBit[2,3], style: Lamp-Lamp1-Red
    Lamp1 (1050,390 20x20), variable: KR4.bInBit[2,4], style: Lamp-Lamp1-Red
    Lamp1 (1050,435 20x20), variable: KR4.bInBit[2,5], style: Lamp-Lamp1-Red
    Lamp1 (1050,480 20x20), variable: KR4.bInBit[2,6], style: Lamp-Lamp1-Red
    Lamp1 (1050,525 20x20), variable: KR4.bInBit[2,7], style: Lamp-Lamp1-Red
    Group (850,10 200x50)
        Button (0,0 200x50), "KR4 E.Stop"
            toggle KR4.KR4_Estop
        Lamp1 (5,5 10x10), variable: KR4.KR4_Estop, style: Lamp-Lamp1-Yellow
    Label (1070,205 110x30), "User Saf"
    Label (1070,250 110x30), "Peri Rdy"
    Label (1070,295 110x30), "IO ActConf"
    Label (1070,340 110x30), "Stop Mess"
    Label (1070,385 110x30), "Pro Act"
    Label (1070,430 110x30), "PGNO Req"
    Label (1070,475 110x30), "Appl Run"
    Label (1070,520 110x30), "Pro Move"
    Label (925,205 105x30), "T1"
    Label (925,250 105x30), "T2"
    Label (925,295 105x30), "Aut"
    Label (925,340 105x30), "Ext"
    Label (925,385 105x30), "On Path"
    Label (925,430 105x30), "In Home"
    Label (925,475 105x30), "RC Rdy1"
    Label (925,520 105x30), "Alarm Stop"
    RoundedRectangle (95,200 110x40), "JIG C Welding"
        toggle KR4.bOutBit[3,0]
    RoundedRectangle (95,245 110x40), "Clean Torch"
        toggle KR4.bOutBit[3,1]
    RoundedRectangle (95,290 110x40), "Go Home"
        toggle KR4.bOutBit[3,2]
    RoundedRectangle (95,335 110x40), "Job Fail"
        toggle KR4.bOutBit[3,3]
    RoundedRectangle (95,380 110x40), "304"
        toggle KR4.bOutBit[3,4]
    RoundedRectangle (95,425 110x40), "305"
        toggle KR4.bOutBit[3,5]
    RoundedRectangle (95,470 110x40), "306"
        toggle KR4.bOutBit[3,6]
    RoundedRectangle (95,515 110x40), "307"
        toggle KR4.bOutBit[3,7]
    Lamp1 (85,210 20x20), variable: KR4.bInBit[3,0], style: Lamp-Lamp1-Red
    Lamp1 (85,255 20x20), variable: KR4.bInBit[3,1], style: Lamp-Lamp1-Red
    Lamp1 (85,300 20x20), variable: KR4.bInBit[3,2], style: Lamp-Lamp1-Red
    Lamp1 (85,345 20x20), variable: KR4.bInBit[3,3], style: Lamp-Lamp1-Red
    Lamp1 (85,390 20x20), variable: KR4.bInBit[3,4], style: Lamp-Lamp1-Red
    Lamp1 (85,435 20x20), variable: KR4.bInBit[3,5], style: Lamp-Lamp1-Red
    Lamp1 (85,480 20x20), variable: KR4.bInBit[3,6], style: Lamp-Lamp1-Red
    Lamp1 (85,525 20x20), variable: KR4.bInBit[3,7], style: Lamp-Lamp1-Red
END_VISUALIZATION

// ---- VISUs/PAGE_KR5.TcVIS
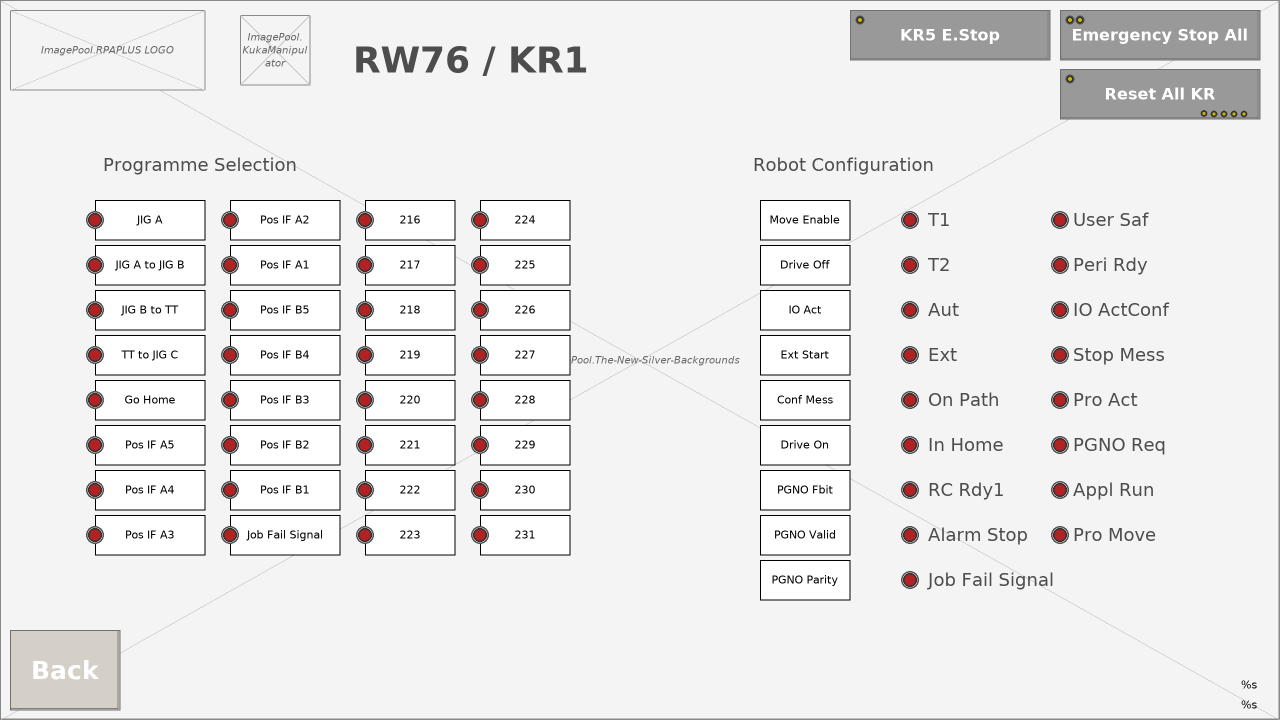
VISUALIZATION PAGE_KR5  // 1280x720
    Image (0,0 1280x720), image: ImagePool.The-New-Silver-Backgrounds
    Frame (0,620 1280x100)
        shows Footer_Back()
    Frame (0,0 1280x150)
        shows Header()
    Label (350,40 300x40), "RW76 / KR1"
    Label (100,150 200x30), "Programme Selection"
    Label (750,150 200x30), "Robot Configuration"
    Lamp1 (900,210 20x20), variable: KR5.bInBit[1,0], style: Lamp-Lamp1-Red
    Lamp1 (900,255 20x20), variable: KR5.bInBit[1,1], style: Lamp-Lamp1-Red
    Lamp1 (900,300 20x20), variable: KR5.bInBit[1,2], style: Lamp-Lamp1-Red
    Lamp1 (900,345 20x20), variable: KR5.bInBit[1,3], style: Lamp-Lamp1-Red
    Lamp1 (900,390 20x20), variable: KR5.bInBit[1,4], style: Lamp-Lamp1-Red
    Lamp1 (900,435 20x20), variable: KR5.bInBit[1,5], style: Lamp-Lamp1-Red
    Lamp1 (900,480 20x20), variable: KR5.bInBit[1,6], style: Lamp-Lamp1-Red
    Lamp1 (900,525 20x20), variable: KR5.bInBit[1,7], style: Lamp-Lamp1-Red
    Lamp1 (1050,210 20x20), variable: KR5.bInBit[2,0], style: Lamp-Lamp1-Red
    Lamp1 (1050,255 20x20), variable: KR5.bInBit[2,1], style: Lamp-Lamp1-Red
    Lamp1 (1050,300 20x20), variable: KR5.bInBit[2,2], style: Lamp-Lamp1-Red
    Lamp1 (1050,345 20x20), variable: KR5.bInBit[2,3], style: Lamp-Lamp1-Red
    Lamp1 (1050,390 20x20), variable: KR5.bInBit[2,4], style: Lamp-Lamp1-Red
    Lamp1 (1050,435 20x20), variable: KR5.bInBit[2,5], style: Lamp-Lamp1-Red
    Lamp1 (1050,480 20x20), variable: KR5.bInBit[2,6], style: Lamp-Lamp1-Red
    Lamp1 (1050,525 20x20), variable: KR5.bInBit[2,7], style: Lamp-Lamp1-Red
    Group (850,10 200x50)
        Button (0,0 200x50), "KR5 E.Stop"
            toggle KR5.KR5_Estop
        Lamp1 (5,5 10x10), variable: KR5.KR5_Estop, style: Lamp-Lamp1-Yellow
    Image (240,15 70x70), image: ImagePool.KukaManipulator
    RoundedRectangle (760,200 90x40), "Move Enable"
        toggle KR5.bOutBit[1,0]
    RoundedRectangle (760,245 90x40), "Drive Off"
        toggle KR5.bOutBit[1,1]
    RoundedRectangle (760,290 90x40), "IO Act"
        toggle KR5.bOutBit[1,2]
    RoundedRectangle (760,335 90x40), "Ext Start"
        toggle KR5.bOutBit[1,3]
    RoundedRectangle (760,380 90x40), "Conf Mess"
        toggle KR5.bOutBit[1,4]
    RoundedRectangle (760,425 90x40), "Drive On"
        toggle KR5.bOutBit[1,5]
    RoundedRectangle (760,470 90x40), "PGNO Fbit"
        toggle KR5.bOutBit[1,6]
    RoundedRectangle (760,515 90x40), "PGNO Valid"
        toggle KR5.bOutBit[1,7]
    RoundedRectangle (760,560 90x40), "PGNO Parity"
        toggle KR5.bOutBit[2,0]
    RoundedRectangle (95,200 110x40), "JIG A"
        toggle KR5.bOutBit[3,0]
    RoundedRectangle (95,245 110x40), "JIG A to JIG B"
        toggle KR5.bOutBit[3,1]
    RoundedRectangle (95,290 110x40), "JIG B to TT"
        toggle KR5.bOutBit[3,2]
    RoundedRectangle (95,335 110x40), "TT to JIG C"
        toggle KR5.bOutBit[3,3]
    RoundedRectangle (95,380 110x40), "Go Home"
        toggle KR5.bOutBit[3,4]
    RoundedRectangle (95,425 110x40), "Pos IF A5"
        toggle KR5.bOutBit[3,5]
    RoundedRectangle (95,470 110x40), "Pos IF A4"
        toggle KR5.bOutBit[3,6]
    RoundedRectangle (95,515 110x40), "Pos IF A3"
        toggle KR5.bOutBit[3,7]
    Label (1070,205 110x30), "User Saf"
    Label (1070,250 110x30), "Peri Rdy"
    Label (1070,295 110x30), "IO ActConf"
    Label (1070,340 110x30), "Stop Mess"
    Label (1070,385 110x30), "Pro Act"
    Label (1070,430 110x30), "PGNO Req"
    Label (1070,475 110x30), "Appl Run"
    Label (1070,520 110x30), "Pro Move"
    Label (925,205 105x30), "T1"
    Label (925,250 105x30), "T2"
    Label (925,295 105x30), "Aut"
    Label (925,340 105x30), "Ext"
    Label (925,385 105x30), "On Path"
    Label (925,430 105x30), "In Home"
    Label (925,475 105x30), "RC Rdy1"
    Label (925,520 105x30), "Alarm Stop"
    Label (925,565 200x30), "Job Fail Signal"
    Lamp1 (900,570 20x20), variable: KR5.bInBit[4,7], style: Lamp-Lamp1-Red
    RoundedRectangle (230,200 110x40), "Pos IF A2"
        toggle KR5.bOutBit[4,0]
    RoundedRectangle (230,245 110x40), "Pos IF A1"
        toggle KR5.bOutBit[4,1]
    RoundedRectangle (230,290 110x40), "Pos IF B5"
        toggle KR5.bOutBit[4,2]
    RoundedRectangle (230,335 110x40), "Pos IF B4"
        toggle KR5.bOutBit[4,3]
    RoundedRectangle (230,380 110x40), "Pos IF B3"
        toggle KR5.bOutBit[4,4]
    RoundedRectangle (230,425 110x40), "Pos IF B2"
        toggle KR5.bOutBit[4,5]
    RoundedRectangle (230,470 110x40), "Pos IF B1"
        toggle KR5.bOutBit[4,6]
    RoundedRectangle (230,515 110x40), "Job Fail Signal"
        toggle KR5.bOutBit[4,7]
    RoundedRectangle (480,200 90x40), "224"
        toggle KR5.bOutBit[6,0]
    RoundedRectangle (480,245 90x40), "225"
        toggle KR5.bOutBit[6,1]
    RoundedRectangle (480,290 90x40), "226"
        toggle KR5.bOutBit[6,2]
    RoundedRectangle (480,335 90x40), "227"
        toggle KR5.bOutBit[6,3]
    RoundedRectangle (480,380 90x40), "228"
        toggle KR5.bOutBit[6,4]
    RoundedRectangle (480,425 90x40), "229"
        toggle KR5.bOutBit[6,5]
    RoundedRectangle (480,470 90x40), "230"
        toggle KR5.bOutBit[6,6]
    RoundedRectangle (480,515 90x40), "231"
        toggle KR5.bOutBit[6,7]
    Lamp1 (470,210 20x20), variable: KR5.bInBit[6,0], style: Lamp-Lamp1-Red
    Lamp1 (470,255 20x20), variable: KR5.bInBit[6,1], style: Lamp-Lamp1-Red
    Lamp1 (470,300 20x20), variable: KR5.bInBit[6,2], style: Lamp-Lamp1-Red
    Lamp1 (470,345 20x20), variable: KR5.bInBit[6,3], style: Lamp-Lamp1-Red
    Lamp1 (470,390 20x20), variable: KR5.bInBit[6,4], style: Lamp-Lamp1-Red
    Lamp1 (470,435 20x20), variable: KR5.bInBit[6,5], style: Lamp-Lamp1-Red
    Lamp1 (470,480 20x20), variable: KR5.bInBit[6,6], style: Lamp-Lamp1-Red
    Lamp1 (470,525 20x20), variable: KR5.bInBit[6,7], style: Lamp-Lamp1-Red
    RoundedRectangle (365,200 90x40), "216"
        toggle KR5.bOutBit[5,0]
    RoundedRectangle (365,245 90x40), "217"
        toggle KR5.bOutBit[5,1]
    RoundedRectangle (365,290 90x40), "218"
        toggle KR5.bOutBit[5,2]
    RoundedRectangle (365,335 90x40), "219"
        toggle KR5.bOutBit[5,3]
    RoundedRectangle (365,380 90x40), "220"
        toggle KR5.bOutBit[5,4]
    RoundedRectangle (365,425 90x40), "221"
        toggle KR5.bOutBit[5,5]
    RoundedRectangle (365,470 90x40), "222"
        toggle KR5.bOutBit[5,6]
    RoundedRectangle (365,515 90x40), "223"
        toggle KR5.bOutBit[5,7]
    Lamp1 (355,210 20x20), variable: KR5.bInBit[5,0], style: Lamp-Lamp1-Red
    Lamp1 (355,255 20x20), variable: KR5.bInBit[5,1], style: Lamp-Lamp1-Red
    Lamp1 (355,300 20x20), variable: KR5.bInBit[5,2], style: Lamp-Lamp1-Red
    Lamp1 (355,345 20x20), variable: KR5.bInBit[5,3], style: Lamp-Lamp1-Red
    Lamp1 (355,390 20x20), variable: KR5.bInBit[5,4], style: Lamp-Lamp1-Red
    Lamp1 (355,435 20x20), variable: KR5.bInBit[5,5], style: Lamp-Lamp1-Red
    Lamp1 (355,480 20x20), variable: KR5.bInBit[5,6], style: Lamp-Lamp1-Red
    Lamp1 (355,525 20x20), variable: KR5.bInBit[5,7], style: Lamp-Lamp1-Red
    Lamp1 (220,210 20x20), variable: KR5.bInBit[4,0], style: Lamp-Lamp1-Red
    Lamp1 (220,255 20x20), variable: KR5.bInBit[4,1], style: Lamp-Lamp1-Red
    Lamp1 (220,300 20x20), variable: KR5.bInBit[4,2], style: Lamp-Lamp1-Red
    Lamp1 (220,345 20x20), variable: KR5.bInBit[4,3], style: Lamp-Lamp1-Red
    Lamp1 (220,390 20x20), variable: KR5.bInBit[4,4], style: Lamp-Lamp1-Red
    Lamp1 (220,435 20x20), variable: KR5.bInBit[4,5], style: Lamp-Lamp1-Red
    Lamp1 (220,480 20x20), variable: KR5.bInBit[4,6], style: Lamp-Lamp1-Red
    Lamp1 (220,525 20x20), variable: KR5.bInBit[4,7], style: Lamp-Lamp1-Red
    Lamp1 (85,210 20x20), variable: KR5.bInBit[3,0], style: Lamp-Lamp1-Red
    Lamp1 (85,255 20x20), variable: KR5.bInBit[3,1], style: Lamp-Lamp1-Red
    Lamp1 (85,300 20x20), variable: KR5.bInBit[3,2], style: Lamp-Lamp1-Red
    Lamp1 (85,345 20x20), variable: KR5.bInBit[3,3], style: Lamp-Lamp1-Red
    Lamp1 (85,390 20x20), variable: KR5.bInBit[3,4], style: Lamp-Lamp1-Red
    Lamp1 (85,435 20x20), variable: KR5.bInBit[3,5], style: Lamp-Lamp1-Red
    Lamp1 (85,480 20x20), variable: KR5.bInBit[3,6], style: Lamp-Lamp1-Red
    Lamp1 (85,525 20x20), variable: KR5.bInBit[3,7], style: Lamp-Lamp1-Red
END_VISUALIZATION

// ---- VISUs/PAGE_KR1.TcVIS
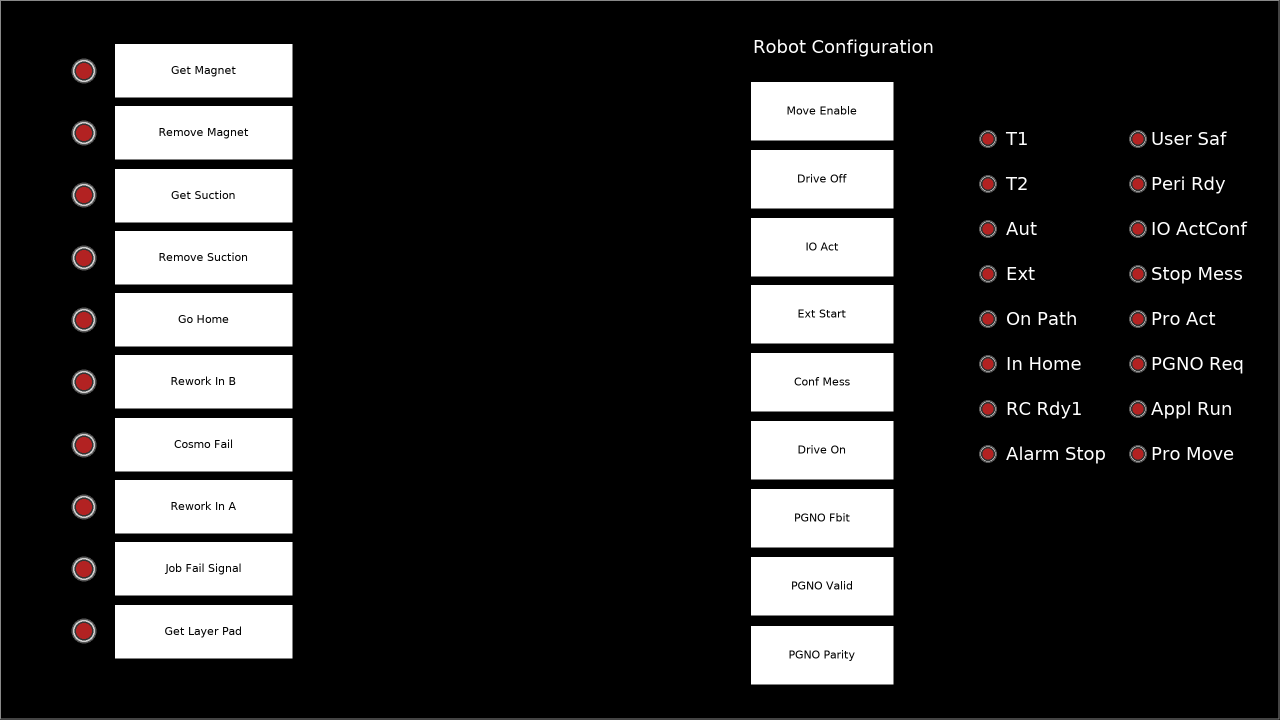
VISUALIZATION PAGE_KR1  // 1280x720
    Lamp1 (64,57 40x28), variable: KR1.bInBit[3,0], style: Lamp-Lamp1-Red
    Lamp1 (64,119 40x28), variable: KR1.bInBit[3,1], style: Lamp-Lamp1-Red
    Lamp1 (64,181 40x28), variable: KR1.bInBit[3,2], style: Lamp-Lamp1-Red
    Lamp1 (64,244 40x28), variable: KR1.bInBit[3,3], style: Lamp-Lamp1-Red
    Lamp1 (64,306 40x28), variable: KR1.bInBit[3,4], style: Lamp-Lamp1-Red
    Lamp1 (64,368 40x28), variable: KR1.bInBit[3,5], style: Lamp-Lamp1-Red
    Lamp1 (64,431 40x28), variable: KR1.bInBit[3,6], style: Lamp-Lamp1-Red
    Lamp1 (64,493 40x28), variable: KR1.bInBit[3,7], style: Lamp-Lamp1-Red
    RoundedRectangle (114,43 179x55), "Get Magnet"
        toggle KR1.bOutBit[3,0]
        OnMouseClick: execute { GVL.KR1_EOAT_FILL := true; }
    RoundedRectangle (114,105 179x55), "Remove Magnet"
        toggle KR1.bOutBit[3,1]
        OnMouseClick: execute { GVL.KR1_EOAT_FILL := false; }
    RoundedRectangle (114,168 179x55), "Get Suction"
        toggle KR1.bOutBit[3,2]
        OnMouseClick: execute { GVL.KR1_EOAT_SUCTION := true; }
    RoundedRectangle (114,230 179x55), "Remove Suction"
        toggle KR1.bOutBit[3,3]
        OnMouseClick: execute { GVL.KR1_EOAT_SUCTION := false; }
    RoundedRectangle (114,292 179x55), "Go Home"
        toggle KR1.bOutBit[3,4]
        OnMouseClick: execute {  }
    RoundedRectangle (114,354 179x55), "Rework In B"
        toggle KR1.bOutBit[3,5]
        OnMouseClick: execute {  }
    RoundedRectangle (114,417 179x55), "Cosmo Fail"
        toggle KR1.bOutBit[3,6]
        OnMouseClick: execute {  }
    RoundedRectangle (114,479 179x55), "Rework In A"
        toggle KR1.bOutBit[3,7]
        OnMouseClick: execute {  }
    RoundedRectangle (114,541 179x55), "Job Fail Signal"
        toggle KR1.bOutBit[4,0]
        OnMouseClick: execute {  }
    RoundedRectangle (114,604 179x55), "Get Layer Pad"
        toggle KR1.bOutBit[4,1]
        OnMouseClick: execute {  }
    Lamp1 (64,555 40x28), variable: KR1.bInBit[4,0], style: Lamp-Lamp1-Red
    Lamp1 (64,617 40x28), variable: KR1.bInBit[4,1], style: Lamp-Lamp1-Red
    RoundedRectangle (750,81 144x60), "Move Enable"
        toggle KR1.bOutBit[1,0]
        OnMouseClick: execute {  }
    RoundedRectangle (750,149 144x60), "Drive Off"
        toggle KR1.bOutBit[1,1]
        OnMouseClick: execute {  }
    RoundedRectangle (750,217 144x60), "IO Act"
        toggle KR1.bOutBit[1,2]
        OnMouseClick: execute {  }
    RoundedRectangle (750,284 144x60), "Ext Start"
        toggle KR1.bOutBit[1,3]
        OnMouseClick: execute {  }
    RoundedRectangle (750,352 144x60), "Conf Mess"
        toggle KR1.bOutBit[1,4]
        OnMouseClick: execute {  }
    RoundedRectangle (750,420 144x60), "Drive On"
        toggle KR1.bOutBit[1,5]
        OnMouseClick: execute {  }
    RoundedRectangle (750,488 144x60), "PGNO Fbit"
        toggle KR1.bOutBit[1,6]
        OnMouseClick: execute {  }
    RoundedRectangle (750,556 144x60), "PGNO Valid"
        toggle KR1.bOutBit[1,7]
        OnMouseClick: execute {  }
    RoundedRectangle (750,625 144x60), "PGNO Parity"
        toggle KR1.bOutBit[2,0]
        OnMouseClick: execute {  }
    Lamp1 (978,129 20x20), variable: KR1.bInBit[1,0], style: Lamp-Lamp1-Red
    Lamp1 (978,174 20x20), variable: KR1.bInBit[1,1], style: Lamp-Lamp1-Red
    Lamp1 (978,219 20x20), variable: KR1.bInBit[1,2], style: Lamp-Lamp1-Red
    Lamp1 (978,264 20x20), variable: KR1.bInBit[1,3], style: Lamp-Lamp1-Red
    Lamp1 (978,309 20x20), variable: KR1.bInBit[1,4], style: Lamp-Lamp1-Red
    Lamp1 (978,354 20x20), variable: KR1.bInBit[1,5], style: Lamp-Lamp1-Red
    Lamp1 (978,399 20x20), variable: KR1.bInBit[1,6], style: Lamp-Lamp1-Red
    Lamp1 (978,444 20x20), variable: KR1.bInBit[1,7], style: Lamp-Lamp1-Red
    Label (1003,124 105x30), "T1"
    Label (1003,169 105x30), "T2"
    Label (1003,214 105x30), "Aut"
    Label (1003,259 105x30), "Ext"
    Label (1003,304 105x30), "On Path"
    Label (1003,349 105x30), "In Home"
    Label (1003,394 105x30), "RC Rdy1"
    Label (1003,439 105x30), "Alarm Stop"
    Lamp1 (1128,129 20x20), variable: KR1.bInBit[2,0], style: Lamp-Lamp1-Red
    Lamp1 (1128,174 20x20), variable: KR1.bInBit[2,1], style: Lamp-Lamp1-Red
    Lamp1 (1128,219 20x20), variable: KR1.bInBit[2,2], style: Lamp-Lamp1-Red
    Lamp1 (1128,264 20x20), variable: KR1.bInBit[2,3], style: Lamp-Lamp1-Red
    Lamp1 (1128,309 20x20), variable: KR1.bInBit[2,4], style: Lamp-Lamp1-Red
    Lamp1 (1128,354 20x20), variable: KR1.bInBit[2,5], style: Lamp-Lamp1-Red
    Lamp1 (1128,399 20x20), variable: KR1.bInBit[2,6], style: Lamp-Lamp1-Red
    Lamp1 (1128,444 20x20), variable: KR1.bInBit[2,7], style: Lamp-Lamp1-Red
    Label (1148,124 110x30), "User Saf"
    Label (1148,169 110x30), "Peri Rdy"
    Label (1148,214 110x30), "IO ActConf"
    Label (1148,259 110x30), "Stop Mess"
    Label (1148,304 110x30), "Pro Act"
    Label (1148,349 110x30), "PGNO Req"
    Label (1148,394 110x30), "Appl Run"
    Label (1148,439 110x30), "Pro Move"
    Label (750,32 250x30), "Robot Configuration"
END_VISUALIZATION
